// TIA Portal V19 export
FUNCTION "SUGAR" : Void   // FC21, LAD
{ S7_Optimized_Access := 'TRUE' }
// stored: SetENOAutomatically false
   VAR_TEMP   // added for the SCL form of the ladder/FBD networks
      _w1 : Bool;
   END_VAR
BEGIN

REGION Network 1: START MFG PROCESS
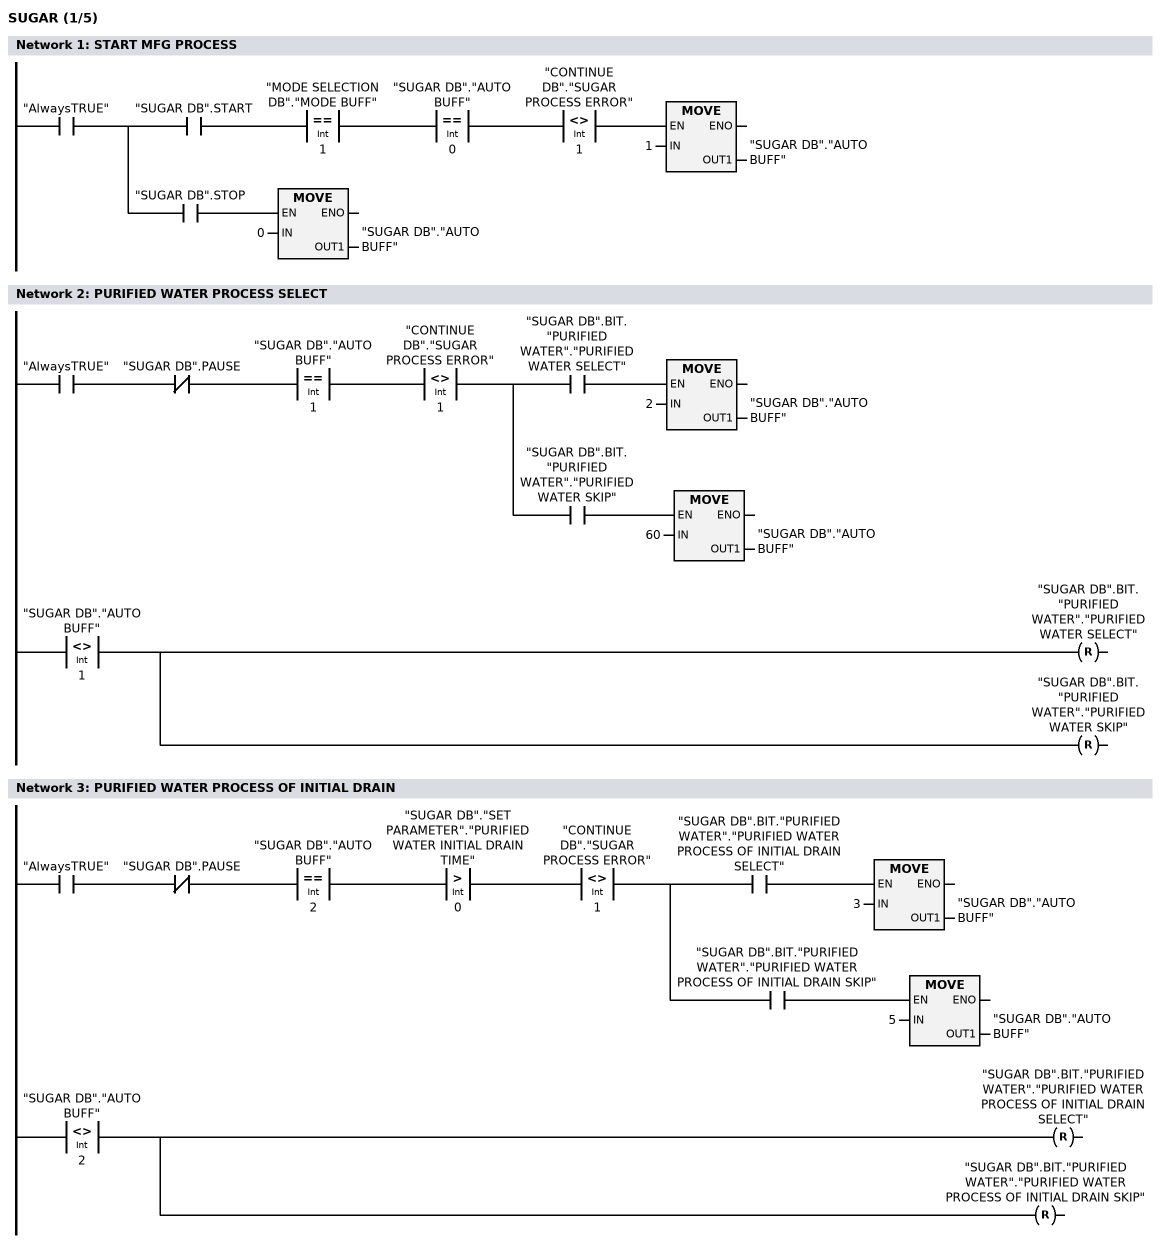
   RUNG wire#powerrail
      Contact( "AlwaysTRUE" )
      wire#w1
      Contact( "SUGAR DB".START )
      { S7_Templates := "SrcType := Int" } EQ_Contact(in1 := "MODE SELECTION DB"."MODE BUFF", in2 := 1)
      { S7_Templates := "SrcType := Int" } EQ_Contact(in1 := "SUGAR DB"."AUTO BUFF", in2 := 0)
      { S7_Templates := "SrcType := Int" } NE_Contact(in1 := "CONTINUE DB"."SUGAR PROCESS ERROR", in2 := 1)
      Move(in := 1, out1 => "SUGAR DB"."AUTO BUFF")
   END_RUNG
   RUNG wire#w1
      Contact( "SUGAR DB".STOP )
      Move(in := 0, out1 => "SUGAR DB"."AUTO BUFF")
   END_RUNG
   // the same network as SCL:
   IF "AlwaysTRUE" AND "SUGAR DB".START AND ("MODE SELECTION DB"."MODE BUFF" = 1) AND ("SUGAR DB"."AUTO BUFF" = 0) AND ("CONTINUE DB"."SUGAR PROCESS ERROR" <> 1) THEN
       "SUGAR DB"."AUTO BUFF" := 1;
   END_IF;
   IF "AlwaysTRUE" AND "SUGAR DB".STOP THEN "SUGAR DB"."AUTO BUFF" := 0; END_IF;
END_REGION

REGION Network 2: PURIFIED WATER PROCESS SELECT
   RUNG wire#powerrail
      Contact( "AlwaysTRUE" )
      I_Contact( "SUGAR DB".PAUSE )
      { S7_Templates := "SrcType := Int" } EQ_Contact(in1 := "SUGAR DB"."AUTO BUFF", in2 := 1)
      { S7_Templates := "SrcType := Int" } NE_Contact(in1 := "CONTINUE DB"."SUGAR PROCESS ERROR", in2 := 1)
      wire#w1
      Contact( "SUGAR DB".BIT."PURIFIED WATER"."PURIFIED WATER SELECT" )
      Move(in := 2, out1 => "SUGAR DB"."AUTO BUFF")
   END_RUNG
   RUNG wire#w1
      Contact( "SUGAR DB".BIT."PURIFIED WATER"."PURIFIED WATER SKIP" )
      Move(in := 60, out1 => "SUGAR DB"."AUTO BUFF")
   END_RUNG
   RUNG wire#powerrail
      { S7_Templates := "SrcType := Int" } NE_Contact(in1 := "SUGAR DB"."AUTO BUFF", in2 := 1)
      wire#w2
      R_Coil( "SUGAR DB".BIT."PURIFIED WATER"."PURIFIED WATER SELECT" )
   END_RUNG
   RUNG wire#w2
      R_Coil( "SUGAR DB".BIT."PURIFIED WATER"."PURIFIED WATER SKIP" )
   END_RUNG
   // the same network as SCL:
   #_w1 := "AlwaysTRUE" AND NOT "SUGAR DB".PAUSE AND ("SUGAR DB"."AUTO BUFF" = 1) AND ("CONTINUE DB"."SUGAR PROCESS ERROR" <> 1);
   IF #_w1 AND "SUGAR DB".BIT."PURIFIED WATER"."PURIFIED WATER SELECT" THEN
       "SUGAR DB"."AUTO BUFF" := 2;
   END_IF;
   IF #_w1 AND "SUGAR DB".BIT."PURIFIED WATER"."PURIFIED WATER SKIP" THEN
       "SUGAR DB"."AUTO BUFF" := 60;
   END_IF;
   IF "SUGAR DB"."AUTO BUFF" <> 1 THEN
       "SUGAR DB".BIT."PURIFIED WATER"."PURIFIED WATER SELECT" := FALSE;
       "SUGAR DB".BIT."PURIFIED WATER"."PURIFIED WATER SKIP" := FALSE;
   END_IF;
END_REGION

REGION Network 3: PURIFIED WATER PROCESS OF INITIAL DRAIN
   RUNG wire#powerrail
      Contact( "AlwaysTRUE" )
      I_Contact( "SUGAR DB".PAUSE )
      { S7_Templates := "SrcType := Int" } EQ_Contact(in1 := "SUGAR DB"."AUTO BUFF", in2 := 2)
      { S7_Templates := "SrcType := Int" } GT_Contact(in1 := "SUGAR DB"."SET PARAMETER"."PURIFIED WATER INITIAL DRAIN TIME", in2 := 0)
      { S7_Templates := "SrcType := Int" } NE_Contact(in1 := "CONTINUE DB"."SUGAR PROCESS ERROR", in2 := 1)
      wire#w1
      Contact( "SUGAR DB".BIT."PURIFIED WATER"."PURIFIED WATER PROCESS OF INITIAL DRAIN SELECT" )
      Move(in := 3, out1 => "SUGAR DB"."AUTO BUFF")
   END_RUNG
   RUNG wire#w1
      Contact( "SUGAR DB".BIT."PURIFIED WATER"."PURIFIED WATER PROCESS OF INITIAL DRAIN SKIP" )
      Move(in := 5, out1 => "SUGAR DB"."AUTO BUFF")
   END_RUNG
   RUNG wire#powerrail
      { S7_Templates := "SrcType := Int" } NE_Contact(in1 := "SUGAR DB"."AUTO BUFF", in2 := 2)
      wire#w2
      R_Coil( "SUGAR DB".BIT."PURIFIED WATER"."PURIFIED WATER PROCESS OF INITIAL DRAIN SELECT" )
   END_RUNG
   RUNG wire#w2
      R_Coil( "SUGAR DB".BIT."PURIFIED WATER"."PURIFIED WATER PROCESS OF INITIAL DRAIN SKIP" )
   END_RUNG
   // the same network as SCL:
   #_w1 := "AlwaysTRUE" AND NOT "SUGAR DB".PAUSE AND ("SUGAR DB"."AUTO BUFF" = 2) AND ("SUGAR DB"."SET PARAMETER"."PURIFIED WATER INITIAL DRAIN TIME" > 0) AND ("CONTINUE DB"."SUGAR PROCESS ERROR" <> 1);
   IF #_w1 AND "SUGAR DB".BIT."PURIFIED WATER"."PURIFIED WATER PROCESS OF INITIAL DRAIN SELECT" THEN
       "SUGAR DB"."AUTO BUFF" := 3;
   END_IF;
   IF #_w1 AND "SUGAR DB".BIT."PURIFIED WATER"."PURIFIED WATER PROCESS OF INITIAL DRAIN SKIP" THEN
       "SUGAR DB"."AUTO BUFF" := 5;
   END_IF;
   IF "SUGAR DB"."AUTO BUFF" <> 2 THEN
       "SUGAR DB".BIT."PURIFIED WATER"."PURIFIED WATER PROCESS OF INITIAL DRAIN SELECT" := FALSE;
       "SUGAR DB".BIT."PURIFIED WATER"."PURIFIED WATER PROCESS OF INITIAL DRAIN SKIP" := FALSE;
   END_IF;
END_REGION

REGION Network 4: TIMER
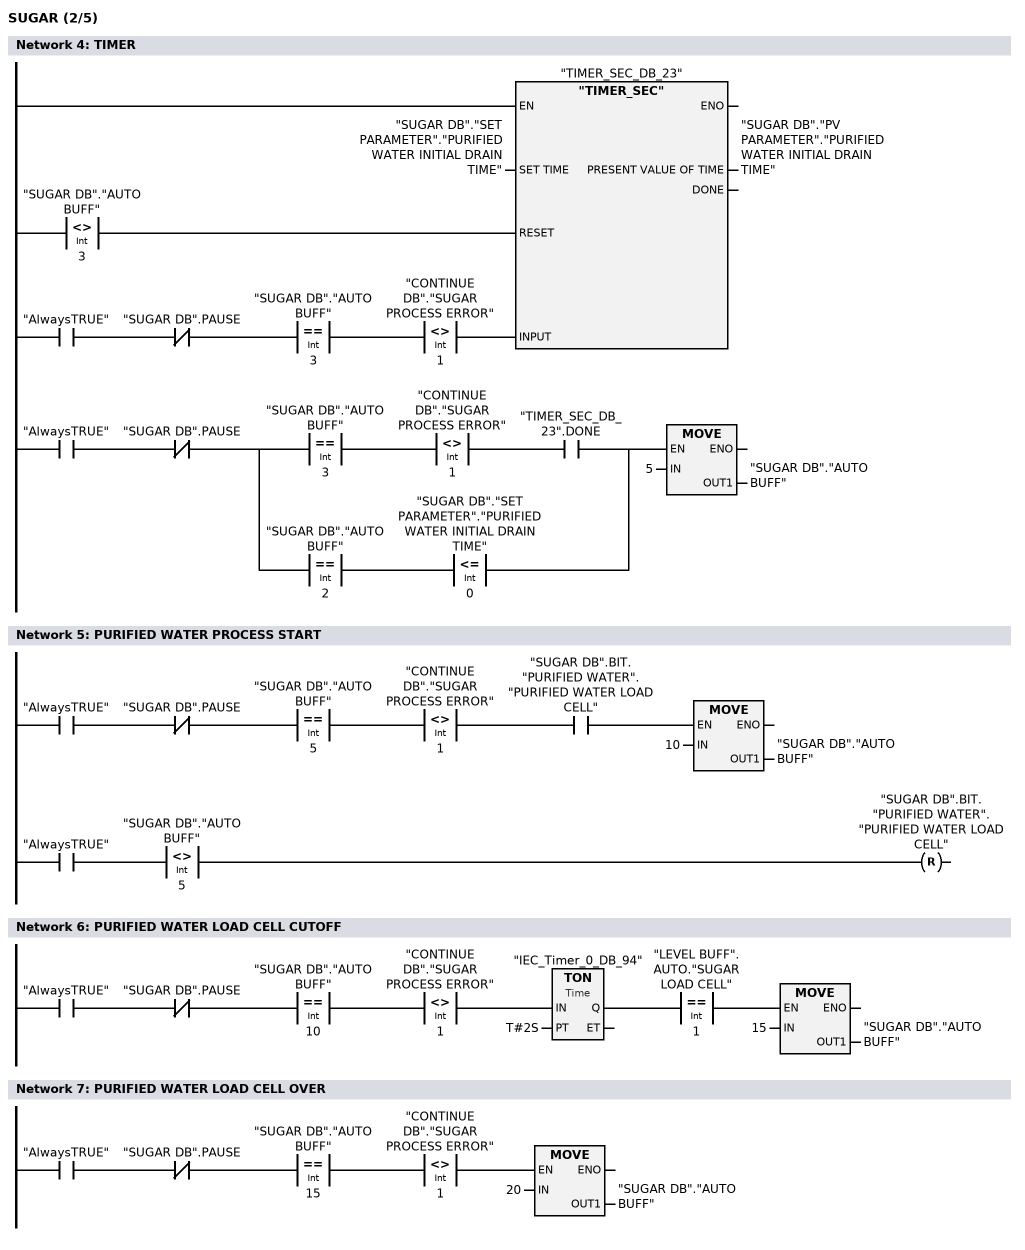
   RUNG wire#powerrail
      "TIMER_SEC_DB_23"(RESET := wire#w1, INPUT := wire#w2, "SET TIME" := "SUGAR DB"."SET PARAMETER"."PURIFIED WATER INITIAL DRAIN TIME", "PRESENT VALUE OF TIME" => "SUGAR DB"."PV PARAMETER"."PURIFIED WATER INITIAL DRAIN TIME", DONE =>)
   END_RUNG
   RUNG wire#powerrail
      { S7_Templates := "SrcType := Int" } NE_Contact(in1 := "SUGAR DB"."AUTO BUFF", in2 := 3)
   END_RUNG wire#w1
   RUNG wire#powerrail
      Contact( "AlwaysTRUE" )
      I_Contact( "SUGAR DB".PAUSE )
      { S7_Templates := "SrcType := Int" } EQ_Contact(in1 := "SUGAR DB"."AUTO BUFF", in2 := 3)
      { S7_Templates := "SrcType := Int" } NE_Contact(in1 := "CONTINUE DB"."SUGAR PROCESS ERROR", in2 := 1)
   END_RUNG wire#w2
   RUNG wire#powerrail
      Contact( "AlwaysTRUE" )
      I_Contact( "SUGAR DB".PAUSE )
      wire#w3
      { S7_Templates := "SrcType := Int" } EQ_Contact(in1 := "SUGAR DB"."AUTO BUFF", in2 := 3)
      { S7_Templates := "SrcType := Int" } NE_Contact(in1 := "CONTINUE DB"."SUGAR PROCESS ERROR", in2 := 1)
      Contact( "TIMER_SEC_DB_23".DONE )
      wire#w4
      Move(in := 5, out1 => "SUGAR DB"."AUTO BUFF")
   END_RUNG
   RUNG wire#w3
      { S7_Templates := "SrcType := Int" } EQ_Contact(in1 := "SUGAR DB"."AUTO BUFF", in2 := 2)
      { S7_Templates := "SrcType := Int" } LE_Contact(in1 := "SUGAR DB"."SET PARAMETER"."PURIFIED WATER INITIAL DRAIN TIME", in2 := 0)
   END_RUNG wire#w4
   // the same network as SCL:
   "TIMER_SEC_DB_23"("SET TIME" := "SUGAR DB"."SET PARAMETER"."PURIFIED WATER INITIAL DRAIN TIME",   // "TIMER_SEC"
                     RESET := "SUGAR DB"."AUTO BUFF" <> 3,
                     INPUT := "AlwaysTRUE" AND NOT "SUGAR DB".PAUSE AND ("SUGAR DB"."AUTO BUFF" = 3) AND ("CONTINUE DB"."SUGAR PROCESS ERROR" <> 1),
                     "PRESENT VALUE OF TIME" => "SUGAR DB"."PV PARAMETER"."PURIFIED WATER INITIAL DRAIN TIME");
   IF "AlwaysTRUE" AND NOT "SUGAR DB".PAUSE AND ((("SUGAR DB"."AUTO BUFF" = 3) AND ("CONTINUE DB"."SUGAR PROCESS ERROR" <> 1) AND "TIMER_SEC_DB_23".DONE) OR (("SUGAR DB"."AUTO BUFF" = 2) AND ("SUGAR DB"."SET PARAMETER"."PURIFIED WATER INITIAL DRAIN TIME" <= 0))) THEN
       "SUGAR DB"."AUTO BUFF" := 5;
   END_IF;
END_REGION

REGION Network 5: PURIFIED WATER PROCESS START
   RUNG wire#powerrail
      Contact( "AlwaysTRUE" )
      I_Contact( "SUGAR DB".PAUSE )
      { S7_Templates := "SrcType := Int" } EQ_Contact(in1 := "SUGAR DB"."AUTO BUFF", in2 := 5)
      { S7_Templates := "SrcType := Int" } NE_Contact(in1 := "CONTINUE DB"."SUGAR PROCESS ERROR", in2 := 1)
      Contact( "SUGAR DB".BIT."PURIFIED WATER"."PURIFIED WATER LOAD CELL" )
      Move(in := 10, out1 => "SUGAR DB"."AUTO BUFF")
   END_RUNG
   RUNG wire#powerrail
      Contact( "AlwaysTRUE" )
      { S7_Templates := "SrcType := Int" } NE_Contact(in1 := "SUGAR DB"."AUTO BUFF", in2 := 5)
      R_Coil( "SUGAR DB".BIT."PURIFIED WATER"."PURIFIED WATER LOAD CELL" )
   END_RUNG
   // the same network as SCL:
   IF "AlwaysTRUE" AND NOT "SUGAR DB".PAUSE AND ("SUGAR DB"."AUTO BUFF" = 5) AND ("CONTINUE DB"."SUGAR PROCESS ERROR" <> 1) AND "SUGAR DB".BIT."PURIFIED WATER"."PURIFIED WATER LOAD CELL" THEN
       "SUGAR DB"."AUTO BUFF" := 10;
   END_IF;
   IF "AlwaysTRUE" AND ("SUGAR DB"."AUTO BUFF" <> 5) THEN
       "SUGAR DB".BIT."PURIFIED WATER"."PURIFIED WATER LOAD CELL" := FALSE;
   END_IF;
END_REGION

REGION Network 6: PURIFIED WATER LOAD CELL CUTOFF
   RUNG wire#powerrail
      Contact( "AlwaysTRUE" )
      I_Contact( "SUGAR DB".PAUSE )
      { S7_Templates := "SrcType := Int" } EQ_Contact(in1 := "SUGAR DB"."AUTO BUFF", in2 := 10)
      { S7_Templates := "SrcType := Int" } NE_Contact(in1 := "CONTINUE DB"."SUGAR PROCESS ERROR", in2 := 1)
      { S7_Templates := "time_type := Time" } "IEC_Timer_0_DB_94".TON(pt := T#2S, et =>)
      { S7_Templates := "SrcType := Int" } EQ_Contact(in1 := "LEVEL BUFF".AUTO."SUGAR LOAD CELL", in2 := 1)
      Move(in := 15, out1 => "SUGAR DB"."AUTO BUFF")
   END_RUNG
   // the same network as SCL:
   "IEC_Timer_0_DB_94".TON(IN := "AlwaysTRUE" AND NOT "SUGAR DB".PAUSE AND ("SUGAR DB"."AUTO BUFF" = 10) AND ("CONTINUE DB"."SUGAR PROCESS ERROR" <> 1),
                           PT := T#2S);
   IF "IEC_Timer_0_DB_94".Q AND ("LEVEL BUFF".AUTO."SUGAR LOAD CELL" = 1) THEN
       "SUGAR DB"."AUTO BUFF" := 15;
   END_IF;
END_REGION

REGION Network 7: PURIFIED WATER LOAD CELL OVER
   RUNG wire#powerrail
      Contact( "AlwaysTRUE" )
      I_Contact( "SUGAR DB".PAUSE )
      { S7_Templates := "SrcType := Int" } EQ_Contact(in1 := "SUGAR DB"."AUTO BUFF", in2 := 15)
      { S7_Templates := "SrcType := Int" } NE_Contact(in1 := "CONTINUE DB"."SUGAR PROCESS ERROR", in2 := 1)
      Move(in := 20, out1 => "SUGAR DB"."AUTO BUFF")
   END_RUNG
   // the same network as SCL:
   IF "AlwaysTRUE" AND NOT "SUGAR DB".PAUSE AND ("SUGAR DB"."AUTO BUFF" = 15) AND ("CONTINUE DB"."SUGAR PROCESS ERROR" <> 1) THEN
       "SUGAR DB"."AUTO BUFF" := 20;
   END_IF;
END_REGION

REGION Network 8: PURIFIED WATER HEATING OR COOLING SEL
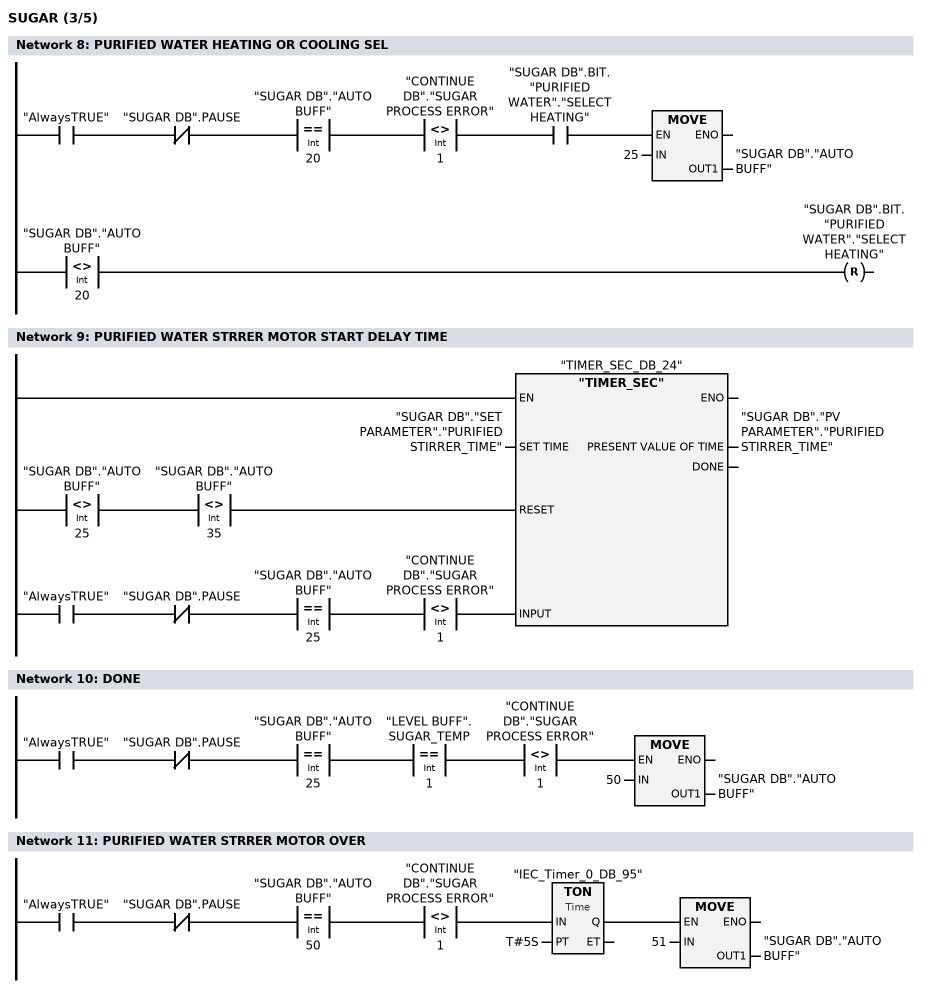
   RUNG wire#powerrail
      Contact( "AlwaysTRUE" )
      I_Contact( "SUGAR DB".PAUSE )
      { S7_Templates := "SrcType := Int" } EQ_Contact(in1 := "SUGAR DB"."AUTO BUFF", in2 := 20)
      { S7_Templates := "SrcType := Int" } NE_Contact(in1 := "CONTINUE DB"."SUGAR PROCESS ERROR", in2 := 1)
      Contact( "SUGAR DB".BIT."PURIFIED WATER"."SELECT HEATING" )
      Move(in := 25, out1 => "SUGAR DB"."AUTO BUFF")
   END_RUNG
   RUNG wire#powerrail
      { S7_Templates := "SrcType := Int" } NE_Contact(in1 := "SUGAR DB"."AUTO BUFF", in2 := 20)
      R_Coil( "SUGAR DB".BIT."PURIFIED WATER"."SELECT HEATING" )
   END_RUNG
   // the same network as SCL:
   IF "AlwaysTRUE" AND NOT "SUGAR DB".PAUSE AND ("SUGAR DB"."AUTO BUFF" = 20) AND ("CONTINUE DB"."SUGAR PROCESS ERROR" <> 1) AND "SUGAR DB".BIT."PURIFIED WATER"."SELECT HEATING" THEN
       "SUGAR DB"."AUTO BUFF" := 25;
   END_IF;
   IF "SUGAR DB"."AUTO BUFF" <> 20 THEN "SUGAR DB".BIT."PURIFIED WATER"."SELECT HEATING" := FALSE; END_IF;
END_REGION

REGION Network 9: PURIFIED WATER STRRER MOTOR START DELAY TIME
   RUNG wire#powerrail
      "TIMER_SEC_DB_24"(RESET := wire#w1, INPUT := wire#w2, "SET TIME" := "SUGAR DB"."SET PARAMETER"."PURIFIED STIRRER_TIME", "PRESENT VALUE OF TIME" => "SUGAR DB"."PV PARAMETER"."PURIFIED STIRRER_TIME", DONE =>)
   END_RUNG
   RUNG wire#powerrail
      { S7_Templates := "SrcType := Int" } NE_Contact(in1 := "SUGAR DB"."AUTO BUFF", in2 := 25)
      { S7_Templates := "SrcType := Int" } NE_Contact(in1 := "SUGAR DB"."AUTO BUFF", in2 := 35)
   END_RUNG wire#w1
   RUNG wire#powerrail
      Contact( "AlwaysTRUE" )
      I_Contact( "SUGAR DB".PAUSE )
      { S7_Templates := "SrcType := Int" } EQ_Contact(in1 := "SUGAR DB"."AUTO BUFF", in2 := 25)
      { S7_Templates := "SrcType := Int" } NE_Contact(in1 := "CONTINUE DB"."SUGAR PROCESS ERROR", in2 := 1)
   END_RUNG wire#w2
   // the same network as SCL:
   "TIMER_SEC_DB_24"("SET TIME" := "SUGAR DB"."SET PARAMETER"."PURIFIED STIRRER_TIME",   // "TIMER_SEC"
                     RESET := ("SUGAR DB"."AUTO BUFF" <> 25) AND ("SUGAR DB"."AUTO BUFF" <> 35),
                     INPUT := "AlwaysTRUE" AND NOT "SUGAR DB".PAUSE AND ("SUGAR DB"."AUTO BUFF" = 25) AND ("CONTINUE DB"."SUGAR PROCESS ERROR" <> 1),
                     "PRESENT VALUE OF TIME" => "SUGAR DB"."PV PARAMETER"."PURIFIED STIRRER_TIME");
END_REGION

REGION Network 10: DONE
   RUNG wire#powerrail
      Contact( "AlwaysTRUE" )
      I_Contact( "SUGAR DB".PAUSE )
      { S7_Templates := "SrcType := Int" } EQ_Contact(in1 := "SUGAR DB"."AUTO BUFF", in2 := 25)
      { S7_Templates := "SrcType := Int" } EQ_Contact(in1 := "LEVEL BUFF".SUGAR_TEMP, in2 := 1)
      { S7_Templates := "SrcType := Int" } NE_Contact(in1 := "CONTINUE DB"."SUGAR PROCESS ERROR", in2 := 1)
      Move(in := 50, out1 => "SUGAR DB"."AUTO BUFF")
   END_RUNG
   // the same network as SCL:
   IF "AlwaysTRUE" AND NOT "SUGAR DB".PAUSE AND ("SUGAR DB"."AUTO BUFF" = 25) AND ("LEVEL BUFF".SUGAR_TEMP = 1) AND ("CONTINUE DB"."SUGAR PROCESS ERROR" <> 1) THEN
       "SUGAR DB"."AUTO BUFF" := 50;
   END_IF;
END_REGION

REGION Network 11: PURIFIED WATER STRRER MOTOR OVER
   RUNG wire#powerrail
      Contact( "AlwaysTRUE" )
      I_Contact( "SUGAR DB".PAUSE )
      { S7_Templates := "SrcType := Int" } EQ_Contact(in1 := "SUGAR DB"."AUTO BUFF", in2 := 50)
      { S7_Templates := "SrcType := Int" } NE_Contact(in1 := "CONTINUE DB"."SUGAR PROCESS ERROR", in2 := 1)
      { S7_Templates := "time_type := Time" } "IEC_Timer_0_DB_95".TON(pt := T#5S, et =>)
      Move(in := 51, out1 => "SUGAR DB"."AUTO BUFF")
   END_RUNG
   // the same network as SCL:
   "IEC_Timer_0_DB_95".TON(IN := "AlwaysTRUE" AND NOT "SUGAR DB".PAUSE AND ("SUGAR DB"."AUTO BUFF" = 50) AND ("CONTINUE DB"."SUGAR PROCESS ERROR" <> 1),
                           PT := T#5S);
   IF "IEC_Timer_0_DB_95".Q THEN "SUGAR DB"."AUTO BUFF" := 51; END_IF;
END_REGION

REGION Network 12: PURIFIED WATER PROCESS OF JACKET DRAIN
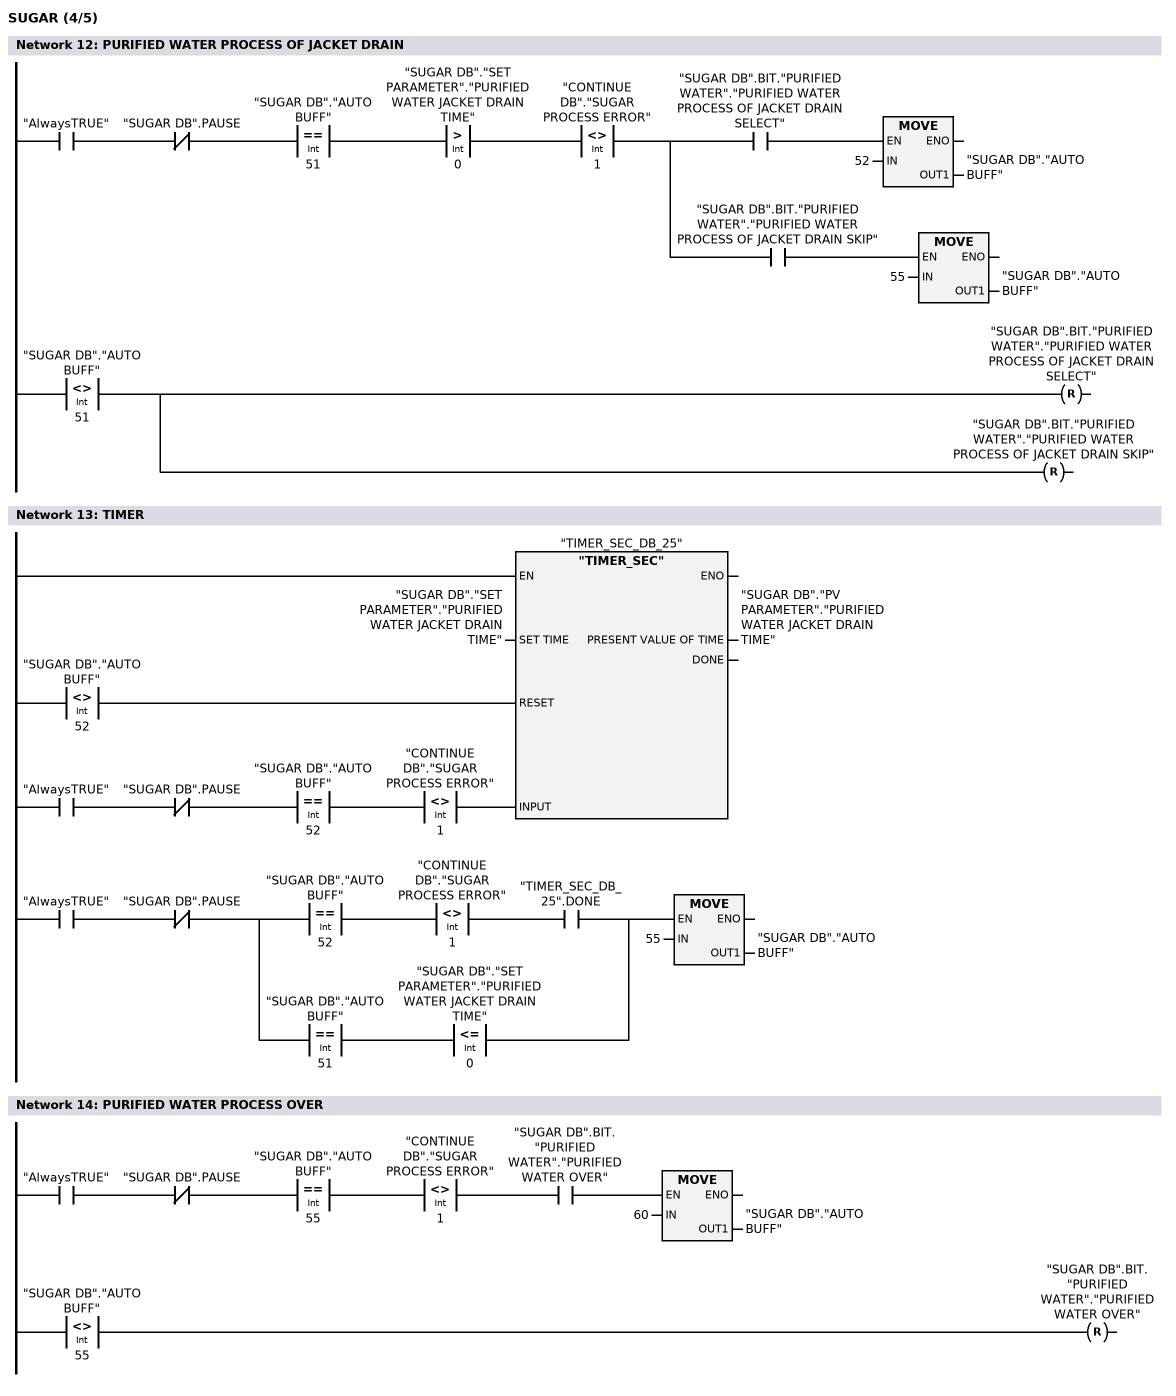
   RUNG wire#powerrail
      Contact( "AlwaysTRUE" )
      I_Contact( "SUGAR DB".PAUSE )
      { S7_Templates := "SrcType := Int" } EQ_Contact(in1 := "SUGAR DB"."AUTO BUFF", in2 := 51)
      { S7_Templates := "SrcType := Int" } GT_Contact(in1 := "SUGAR DB"."SET PARAMETER"."PURIFIED WATER JACKET DRAIN TIME", in2 := 0)
      { S7_Templates := "SrcType := Int" } NE_Contact(in1 := "CONTINUE DB"."SUGAR PROCESS ERROR", in2 := 1)
      wire#w1
      Contact( "SUGAR DB".BIT."PURIFIED WATER"."PURIFIED WATER PROCESS OF JACKET DRAIN SELECT" )
      Move(in := 52, out1 => "SUGAR DB"."AUTO BUFF")
   END_RUNG
   RUNG wire#w1
      Contact( "SUGAR DB".BIT."PURIFIED WATER"."PURIFIED WATER PROCESS OF JACKET DRAIN SKIP" )
      Move(in := 55, out1 => "SUGAR DB"."AUTO BUFF")
   END_RUNG
   RUNG wire#powerrail
      { S7_Templates := "SrcType := Int" } NE_Contact(in1 := "SUGAR DB"."AUTO BUFF", in2 := 51)
      wire#w2
      R_Coil( "SUGAR DB".BIT."PURIFIED WATER"."PURIFIED WATER PROCESS OF JACKET DRAIN SELECT" )
   END_RUNG
   RUNG wire#w2
      R_Coil( "SUGAR DB".BIT."PURIFIED WATER"."PURIFIED WATER PROCESS OF JACKET DRAIN SKIP" )
   END_RUNG
   // the same network as SCL:
   #_w1 := "AlwaysTRUE" AND NOT "SUGAR DB".PAUSE AND ("SUGAR DB"."AUTO BUFF" = 51) AND ("SUGAR DB"."SET PARAMETER"."PURIFIED WATER JACKET DRAIN TIME" > 0) AND ("CONTINUE DB"."SUGAR PROCESS ERROR" <> 1);
   IF #_w1 AND "SUGAR DB".BIT."PURIFIED WATER"."PURIFIED WATER PROCESS OF JACKET DRAIN SELECT" THEN
       "SUGAR DB"."AUTO BUFF" := 52;
   END_IF;
   IF #_w1 AND "SUGAR DB".BIT."PURIFIED WATER"."PURIFIED WATER PROCESS OF JACKET DRAIN SKIP" THEN
       "SUGAR DB"."AUTO BUFF" := 55;
   END_IF;
   IF "SUGAR DB"."AUTO BUFF" <> 51 THEN
       "SUGAR DB".BIT."PURIFIED WATER"."PURIFIED WATER PROCESS OF JACKET DRAIN SELECT" := FALSE;
       "SUGAR DB".BIT."PURIFIED WATER"."PURIFIED WATER PROCESS OF JACKET DRAIN SKIP" := FALSE;
   END_IF;
END_REGION

REGION Network 13: TIMER
   RUNG wire#powerrail
      "TIMER_SEC_DB_25"(RESET := wire#w1, INPUT := wire#w2, "SET TIME" := "SUGAR DB"."SET PARAMETER"."PURIFIED WATER JACKET DRAIN TIME", "PRESENT VALUE OF TIME" => "SUGAR DB"."PV PARAMETER"."PURIFIED WATER JACKET DRAIN TIME", DONE =>)
   END_RUNG
   RUNG wire#powerrail
      { S7_Templates := "SrcType := Int" } NE_Contact(in1 := "SUGAR DB"."AUTO BUFF", in2 := 52)
   END_RUNG wire#w1
   RUNG wire#powerrail
      Contact( "AlwaysTRUE" )
      I_Contact( "SUGAR DB".PAUSE )
      { S7_Templates := "SrcType := Int" } EQ_Contact(in1 := "SUGAR DB"."AUTO BUFF", in2 := 52)
      { S7_Templates := "SrcType := Int" } NE_Contact(in1 := "CONTINUE DB"."SUGAR PROCESS ERROR", in2 := 1)
   END_RUNG wire#w2
   RUNG wire#powerrail
      Contact( "AlwaysTRUE" )
      I_Contact( "SUGAR DB".PAUSE )
      wire#w3
      { S7_Templates := "SrcType := Int" } EQ_Contact(in1 := "SUGAR DB"."AUTO BUFF", in2 := 52)
      { S7_Templates := "SrcType := Int" } NE_Contact(in1 := "CONTINUE DB"."SUGAR PROCESS ERROR", in2 := 1)
      Contact( "TIMER_SEC_DB_25".DONE )
      wire#w4
      Move(in := 55, out1 => "SUGAR DB"."AUTO BUFF")
   END_RUNG
   RUNG wire#w3
      { S7_Templates := "SrcType := Int" } EQ_Contact(in1 := "SUGAR DB"."AUTO BUFF", in2 := 51)
      { S7_Templates := "SrcType := Int" } LE_Contact(in1 := "SUGAR DB"."SET PARAMETER"."PURIFIED WATER JACKET DRAIN TIME", in2 := 0)
   END_RUNG wire#w4
   // the same network as SCL:
   "TIMER_SEC_DB_25"("SET TIME" := "SUGAR DB"."SET PARAMETER"."PURIFIED WATER JACKET DRAIN TIME",   // "TIMER_SEC"
                     RESET := "SUGAR DB"."AUTO BUFF" <> 52,
                     INPUT := "AlwaysTRUE" AND NOT "SUGAR DB".PAUSE AND ("SUGAR DB"."AUTO BUFF" = 52) AND ("CONTINUE DB"."SUGAR PROCESS ERROR" <> 1),
                     "PRESENT VALUE OF TIME" => "SUGAR DB"."PV PARAMETER"."PURIFIED WATER JACKET DRAIN TIME");
   IF "AlwaysTRUE" AND NOT "SUGAR DB".PAUSE AND ((("SUGAR DB"."AUTO BUFF" = 52) AND ("CONTINUE DB"."SUGAR PROCESS ERROR" <> 1) AND "TIMER_SEC_DB_25".DONE) OR (("SUGAR DB"."AUTO BUFF" = 51) AND ("SUGAR DB"."SET PARAMETER"."PURIFIED WATER JACKET DRAIN TIME" <= 0))) THEN
       "SUGAR DB"."AUTO BUFF" := 55;
   END_IF;
END_REGION

REGION Network 14: PURIFIED WATER PROCESS OVER
   RUNG wire#powerrail
      Contact( "AlwaysTRUE" )
      I_Contact( "SUGAR DB".PAUSE )
      { S7_Templates := "SrcType := Int" } EQ_Contact(in1 := "SUGAR DB"."AUTO BUFF", in2 := 55)
      { S7_Templates := "SrcType := Int" } NE_Contact(in1 := "CONTINUE DB"."SUGAR PROCESS ERROR", in2 := 1)
      Contact( "SUGAR DB".BIT."PURIFIED WATER"."PURIFIED WATER OVER" )
      Move(in := 60, out1 => "SUGAR DB"."AUTO BUFF")
   END_RUNG
   RUNG wire#powerrail
      { S7_Templates := "SrcType := Int" } NE_Contact(in1 := "SUGAR DB"."AUTO BUFF", in2 := 55)
      R_Coil( "SUGAR DB".BIT."PURIFIED WATER"."PURIFIED WATER OVER" )
   END_RUNG
   // the same network as SCL:
   IF "AlwaysTRUE" AND NOT "SUGAR DB".PAUSE AND ("SUGAR DB"."AUTO BUFF" = 55) AND ("CONTINUE DB"."SUGAR PROCESS ERROR" <> 1) AND "SUGAR DB".BIT."PURIFIED WATER"."PURIFIED WATER OVER" THEN
       "SUGAR DB"."AUTO BUFF" := 60;
   END_IF;
   IF "SUGAR DB"."AUTO BUFF" <> 55 THEN
       "SUGAR DB".BIT."PURIFIED WATER"."PURIFIED WATER OVER" := FALSE;
   END_IF;
END_REGION

REGION Network 16: MATERIAL SUCTION SELECT / SKIP //////////////////////////////
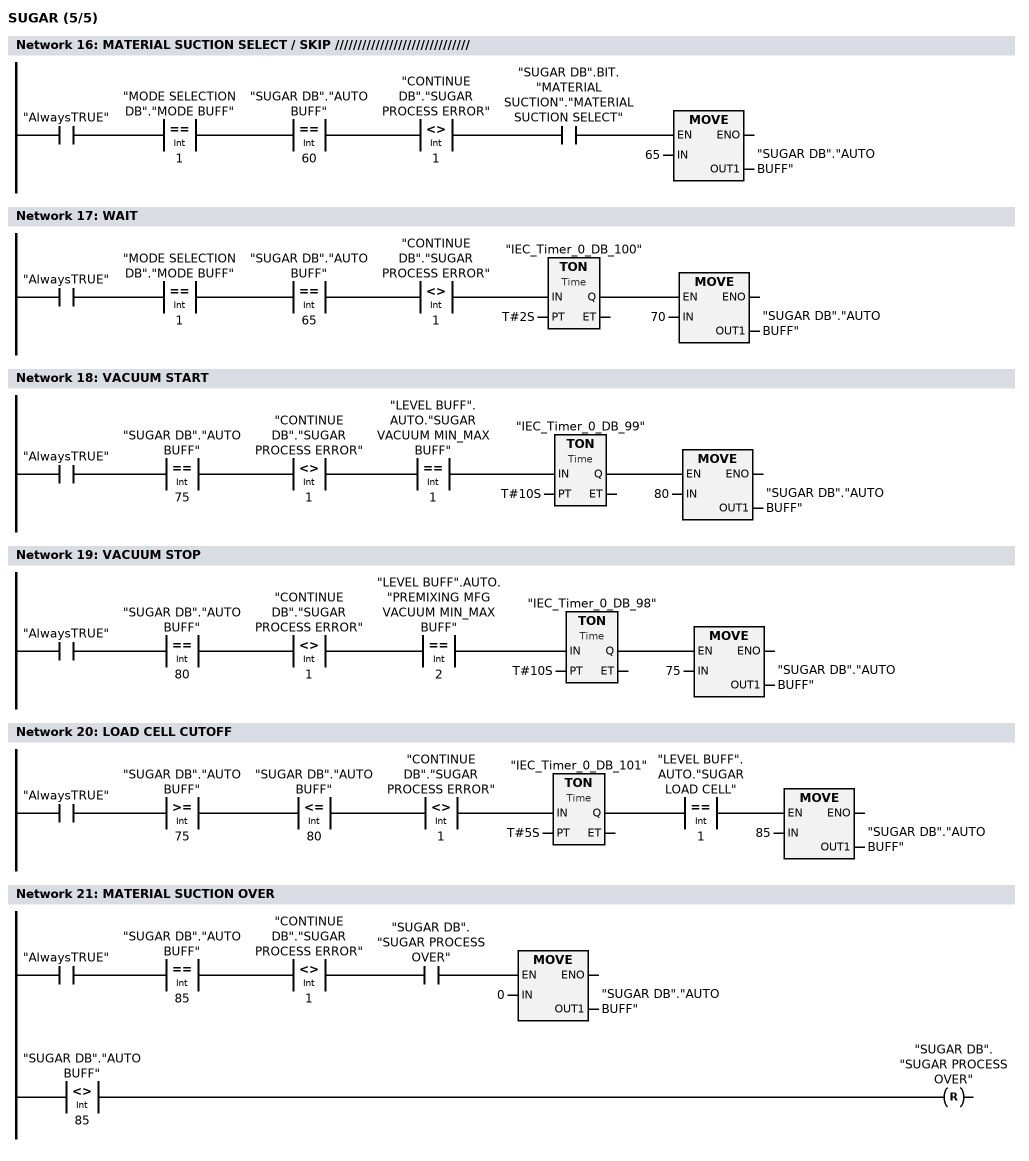
   RUNG wire#powerrail
      Contact( "AlwaysTRUE" )
      { S7_Templates := "SrcType := Int" } EQ_Contact(in1 := "MODE SELECTION DB"."MODE BUFF", in2 := 1)
      { S7_Templates := "SrcType := Int" } EQ_Contact(in1 := "SUGAR DB"."AUTO BUFF", in2 := 60)
      { S7_Templates := "SrcType := Int" } NE_Contact(in1 := "CONTINUE DB"."SUGAR PROCESS ERROR", in2 := 1)
      Contact( "SUGAR DB".BIT."MATERIAL SUCTION"."MATERIAL SUCTION SELECT" )
      Move(in := 65, out1 => "SUGAR DB"."AUTO BUFF")
   END_RUNG
   // the same network as SCL:
   IF "AlwaysTRUE" AND ("MODE SELECTION DB"."MODE BUFF" = 1) AND ("SUGAR DB"."AUTO BUFF" = 60) AND ("CONTINUE DB"."SUGAR PROCESS ERROR" <> 1) AND "SUGAR DB".BIT."MATERIAL SUCTION"."MATERIAL SUCTION SELECT" THEN
       "SUGAR DB"."AUTO BUFF" := 65;
   END_IF;
END_REGION

REGION Network 17: WAIT
   RUNG wire#powerrail
      Contact( "AlwaysTRUE" )
      { S7_Templates := "SrcType := Int" } EQ_Contact(in1 := "MODE SELECTION DB"."MODE BUFF", in2 := 1)
      { S7_Templates := "SrcType := Int" } EQ_Contact(in1 := "SUGAR DB"."AUTO BUFF", in2 := 65)
      { S7_Templates := "SrcType := Int" } NE_Contact(in1 := "CONTINUE DB"."SUGAR PROCESS ERROR", in2 := 1)
      { S7_Templates := "time_type := Time" } "IEC_Timer_0_DB_100".TON(pt := T#2S, et =>)
      Move(in := 70, out1 => "SUGAR DB"."AUTO BUFF")
   END_RUNG
   // the same network as SCL:
   "IEC_Timer_0_DB_100".TON(IN := "AlwaysTRUE" AND ("MODE SELECTION DB"."MODE BUFF" = 1) AND ("SUGAR DB"."AUTO BUFF" = 65) AND ("CONTINUE DB"."SUGAR PROCESS ERROR" <> 1),
                           PT := T#2S);
   IF "IEC_Timer_0_DB_100".Q THEN "SUGAR DB"."AUTO BUFF" := 70; END_IF;
END_REGION

REGION Network 18: VACUUM START
   RUNG wire#powerrail
      Contact( "AlwaysTRUE" )
      { S7_Templates := "SrcType := Int" } EQ_Contact(in1 := "SUGAR DB"."AUTO BUFF", in2 := 75)
      { S7_Templates := "SrcType := Int" } NE_Contact(in1 := "CONTINUE DB"."SUGAR PROCESS ERROR", in2 := 1)
      { S7_Templates := "SrcType := Int" } EQ_Contact(in1 := "LEVEL BUFF".AUTO."SUGAR VACUUM MIN_MAX BUFF", in2 := 1)
      { S7_Templates := "time_type := Time" } "IEC_Timer_0_DB_99".TON(pt := T#10S, et =>)
      Move(in := 80, out1 => "SUGAR DB"."AUTO BUFF")
   END_RUNG
   // the same network as SCL:
   "IEC_Timer_0_DB_99".TON(IN := "AlwaysTRUE" AND ("SUGAR DB"."AUTO BUFF" = 75) AND ("CONTINUE DB"."SUGAR PROCESS ERROR" <> 1) AND ("LEVEL BUFF".AUTO."SUGAR VACUUM MIN_MAX BUFF" = 1),
                           PT := T#10S);
   IF "IEC_Timer_0_DB_99".Q THEN "SUGAR DB"."AUTO BUFF" := 80; END_IF;
END_REGION

REGION Network 19: VACUUM STOP
   RUNG wire#powerrail
      Contact( "AlwaysTRUE" )
      { S7_Templates := "SrcType := Int" } EQ_Contact(in1 := "SUGAR DB"."AUTO BUFF", in2 := 80)
      { S7_Templates := "SrcType := Int" } NE_Contact(in1 := "CONTINUE DB"."SUGAR PROCESS ERROR", in2 := 1)
      { S7_Templates := "SrcType := Int" } EQ_Contact(in1 := "LEVEL BUFF".AUTO."PREMIXING MFG VACUUM MIN_MAX BUFF", in2 := 2)
      { S7_Templates := "time_type := Time" } "IEC_Timer_0_DB_98".TON(pt := T#10S, et =>)
      Move(in := 75, out1 => "SUGAR DB"."AUTO BUFF")
   END_RUNG
   // the same network as SCL:
   "IEC_Timer_0_DB_98".TON(IN := "AlwaysTRUE" AND ("SUGAR DB"."AUTO BUFF" = 80) AND ("CONTINUE DB"."SUGAR PROCESS ERROR" <> 1) AND ("LEVEL BUFF".AUTO."PREMIXING MFG VACUUM MIN_MAX BUFF" = 2),
                           PT := T#10S);
   IF "IEC_Timer_0_DB_98".Q THEN "SUGAR DB"."AUTO BUFF" := 75; END_IF;
END_REGION

REGION Network 20: LOAD CELL CUTOFF
   RUNG wire#powerrail
      Contact( "AlwaysTRUE" )
      { S7_Templates := "SrcType := Int" } GE_Contact(in1 := "SUGAR DB"."AUTO BUFF", in2 := 75)
      { S7_Templates := "SrcType := Int" } LE_Contact(in1 := "SUGAR DB"."AUTO BUFF", in2 := 80)
      { S7_Templates := "SrcType := Int" } NE_Contact(in1 := "CONTINUE DB"."SUGAR PROCESS ERROR", in2 := 1)
      { S7_Templates := "time_type := Time" } "IEC_Timer_0_DB_101".TON(pt := T#5S, et =>)
      { S7_Templates := "SrcType := Int" } EQ_Contact(in1 := "LEVEL BUFF".AUTO."SUGAR LOAD CELL", in2 := 1)
      Move(in := 85, out1 => "SUGAR DB"."AUTO BUFF")
   END_RUNG
   // the same network as SCL:
   "IEC_Timer_0_DB_101".TON(IN := "AlwaysTRUE" AND ("SUGAR DB"."AUTO BUFF" >= 75) AND ("SUGAR DB"."AUTO BUFF" <= 80) AND ("CONTINUE DB"."SUGAR PROCESS ERROR" <> 1),
                           PT := T#5S);
   IF "IEC_Timer_0_DB_101".Q AND ("LEVEL BUFF".AUTO."SUGAR LOAD CELL" = 1) THEN
       "SUGAR DB"."AUTO BUFF" := 85;
   END_IF;
END_REGION

REGION Network 21: MATERIAL SUCTION OVER
   RUNG wire#powerrail
      Contact( "AlwaysTRUE" )
      { S7_Templates := "SrcType := Int" } EQ_Contact(in1 := "SUGAR DB"."AUTO BUFF", in2 := 85)
      { S7_Templates := "SrcType := Int" } NE_Contact(in1 := "CONTINUE DB"."SUGAR PROCESS ERROR", in2 := 1)
      Contact( "SUGAR DB"."SUGAR PROCESS OVER" )
      Move(in := 0, out1 => "SUGAR DB"."AUTO BUFF")
   END_RUNG
   RUNG wire#powerrail
      { S7_Templates := "SrcType := Int" } NE_Contact(in1 := "SUGAR DB"."AUTO BUFF", in2 := 85)
      R_Coil( "SUGAR DB"."SUGAR PROCESS OVER" )
   END_RUNG
   // the same network as SCL:
   IF "AlwaysTRUE" AND ("SUGAR DB"."AUTO BUFF" = 85) AND ("CONTINUE DB"."SUGAR PROCESS ERROR" <> 1) AND "SUGAR DB"."SUGAR PROCESS OVER" THEN
       "SUGAR DB"."AUTO BUFF" := 0;
   END_IF;
   IF "SUGAR DB"."AUTO BUFF" <> 85 THEN "SUGAR DB"."SUGAR PROCESS OVER" := FALSE; END_IF;
END_REGION
END_FUNCTION
